// TIA Portal V20 export
DATA_BLOCK "DB_SystemSimu"   // DB30
// stored: Access Published, MemoryReserve 100, Namespace Global
   VAR
      TriggerSensor : Struct
         Line : Struct
            A1 : Struct
               Conveyor : Array[_.gMinA1.._.gMaxA1] of Bool;
            END_STRUCT;
            B1 : Struct
               Conveyor : Array[_.gMinB1.._.gMaxB1] of Bool;
            END_STRUCT;
            C1 : Struct
               Conveyor : Array[_.gMinC1.._.gMaxC1] of Bool;
            END_STRUCT;
            D1 : Struct
               Conveyor : Array[_.gMinD1.._.gMaxD1] of Bool;
            END_STRUCT;
         END_STRUCT;
      END_STRUCT;
      TriggerFault : Struct
         Line : Struct
            A1 : Struct
               Conveyor : Array[_.gMinA1.._.gMaxA1] of Bool;
            END_STRUCT;
            B1 : Struct
               Conveyor : Array[_.gMinB1.._.gMaxB1] of Bool;
            END_STRUCT;
            C1 : Struct
               Conveyor : Array[_.gMinC1.._.gMaxC1] of Bool;
            END_STRUCT;
            D1 : Struct
               Conveyor : Array[_.gMinD1.._.gMaxD1] of Bool;
            END_STRUCT;
         END_STRUCT;
      END_STRUCT;
      Fire : Bool;
   END_VAR
BEGIN
   // TriggerSensor.Line.A1.Conveyor[1001] : AS1.1.1
   // TriggerSensor.Line.A1.Conveyor[1002] : AS1.1.2
   // TriggerFault.Line.A1.Conveyor[1001] : AS1.1.1
   // TriggerFault.Line.A1.Conveyor[1002] : AS1.1.2
END_DATA_BLOCK
